{attribute 'GeneratedUsingTerminal: EL3443-0000-0016'}
{attribute addProperty BoxType "EL3443-0000-0016"}
{attribute addProperty Id "VoltageAT %I*REAL4CurrentAT %I*REAL4"}
{attribute addProperty CRC "1717073118"}
{attribute addProperty Size "8"}
TYPE L1_Basic_665874DE EXTENDS InputBase_8311D824 :
STRUCT
	{attribute addProperty Name "Voltage"}
	Voltage AT %I* : REAL;
	{attribute addProperty Name "Current"}
	Current AT %I* : REAL;
END_STRUCT
END_TYPE

(* stored: Version 1.2.0.0, ProductVersion 3.1.4024.9
   DUT L1_Basic_665874DE: Id {e857e1b9-31e6-443d-a06c-60e0e2ec38da} *)
